TYPE ST_MeasurementFieldData :
STRUCT
	//Power
	ar_ApparentPower			: 	ARRAY[0..3] OF REAL;
	ar_ReactivePower			: 	ARRAY[0..3] OF REAL;
	ar_ActivePower				: 	ARRAY[0..3] OF REAL;

	//Energy Consumed
	r_EnergyConsumed			:	REAL := 0;
	
	//Energy Delivered
	r_EnergySupplied			:	REAL := 0;
	
	//THD
	ar_THD						:	ARRAY[0..3] OF REAL := [0, 0, 0, 0];	
	
	//PF
	ar_PowerFactor				:	ARRAY[0..3] OF REAL := [0, 0, 0, 0];
	
	//Current
	ar_Current					: 	ARRAY[0..4] OF REAL := [0, 0, 0, 0];
	r_CurrentUnbalance			:	REAL;
END_STRUCT
END_TYPE

(* stored: Version 1.1.0.1, ProductVersion 3.1.4024.12
   DUT ST_MeasurementFieldData: Id {a8bd4a52-8c63-4e9b-912a-3f9213046c82} *)
